// TIA Portal V16 export
// export: Created 2023-01-03T15:54:37.2222121Z, ExportSetting WithDefaults, DisplayName Totally Integrated Automation Portal, DisplayVersion V16, DisplayName TIA Portal Version Control Interface, DisplayVersion V16, DisplayName TIA Portal Openness, DisplayVersion V16, DisplayName STEP 7 Professional, DisplayVersion V16, DisplayName STEP 7 Safety, DisplayVersion V16, DisplayName WinCC Advanced, DisplayVersion V16
FUNCTION_BLOCK "MOTOR_AUTO"   // FB2, LAD
{ S7_Optimized_Access := 'TRUE' }
VERSION : 0.1
// stored: AutoNumber true, IsIECCheckEnabled false, IsRetainMemResEnabled false, MemoryReserve 100, SetENOAutomatically false, UDAEnableTagReadback false
   VAR_TEMP   // added for the SCL form of the ladder/FBD networks
      _w1 : Bool;
      _w2 : Bool;
   END_VAR
BEGIN

REGION Network 1: conveyor motor -M1 forwards fixed speed
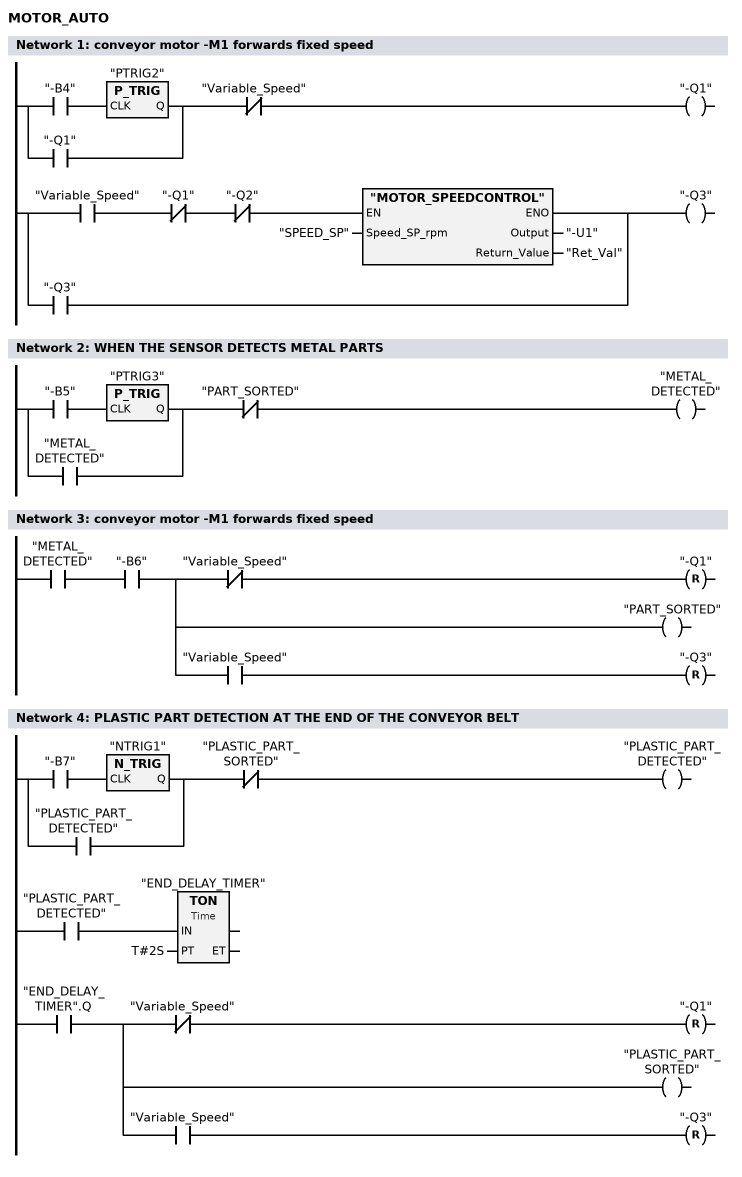
   RUNG wire#powerrail
      Contact( "-B4" )
      P_Trig( "PTRIG2" )
      wire#w1
      I_Contact( "Variable_Speed" )
      Coil( "-Q1" )
   END_RUNG
   RUNG wire#powerrail
      Contact( "-Q1" )
   END_RUNG wire#w1
   RUNG wire#powerrail
      Contact( "Variable_Speed" )
      I_Contact( "-Q1" )
      I_Contact( "-Q2" )
      "MOTOR_SPEEDCONTROL"(Speed_SP_rpm := "SPEED_SP", Output => "-U1", Return_Value => "Ret_Val")
      wire#w2
      Coil( "-Q3" )
   END_RUNG
   RUNG wire#powerrail
      Contact( "-Q3" )
   END_RUNG wire#w2
   // the same network as SCL:
   #_w1 := "-B4" AND NOT "PTRIG2";   // rising edge
   "PTRIG2" := "-B4";
   "-Q1" := (#_w1 OR "-Q1") AND NOT "Variable_Speed";
   "MOTOR_SPEEDCONTROL"(EN := "Variable_Speed" AND NOT "-Q1" AND NOT "-Q2",
                        Speed_SP_rpm := "SPEED_SP",
                        Output => "-U1",
                        Return_Value => "Ret_Val",
                        ENO => #_w2);
   "-Q3" := #_w2 OR "-Q3";
END_REGION

REGION Network 2: WHEN THE SENSOR DETECTS METAL PARTS
   RUNG wire#powerrail
      Contact( "-B5" )
      P_Trig( "PTRIG3" )
      wire#w1
      I_Contact( "PART_SORTED" )
      Coil( "METAL_DETECTED" )
   END_RUNG
   RUNG wire#powerrail
      Contact( "METAL_DETECTED" )
   END_RUNG wire#w1
   // the same network as SCL:
   #_w1 := "-B5" AND NOT "PTRIG3";   // rising edge
   "PTRIG3" := "-B5";
   "METAL_DETECTED" := (#_w1 OR "METAL_DETECTED") AND NOT "PART_SORTED";
END_REGION

REGION Network 3: conveyor motor -M1 forwards fixed speed
   RUNG wire#powerrail
      Contact( "METAL_DETECTED" )
      Contact( "-B6" )
      wire#w1
      I_Contact( "Variable_Speed" )
      R_Coil( "-Q1" )
   END_RUNG
   RUNG wire#w1
      Coil( "PART_SORTED" )
   END_RUNG
   RUNG wire#w1
      Contact( "Variable_Speed" )
      R_Coil( "-Q3" )
   END_RUNG
   // the same network as SCL:
   #_w1 := "METAL_DETECTED" AND "-B6";
   IF #_w1 AND NOT "Variable_Speed" THEN "-Q1" := FALSE; END_IF;
   "PART_SORTED" := #_w1;
   IF #_w1 AND "Variable_Speed" THEN "-Q3" := FALSE; END_IF;
END_REGION

REGION Network 4: PLASTIC PART DETECTION AT THE END OF THE CONVEYOR BELT
   RUNG wire#powerrail
      Contact( "-B7" )
      N_Trig( "NTRIG1" )
      wire#w1
      I_Contact( "PLASTIC_PART_SORTED" )
      Coil( "PLASTIC_PART_DETECTED" )
   END_RUNG
   RUNG wire#powerrail
      Contact( "PLASTIC_PART_DETECTED" )
   END_RUNG wire#w1
   RUNG wire#powerrail
      Contact( "PLASTIC_PART_DETECTED" )
      { S7_Templates := "time_type := Time" } "END_DELAY_TIMER".TON(pt := T#2S, et =>)
   END_RUNG
   RUNG wire#powerrail
      Contact( "END_DELAY_TIMER".Q )
      wire#w2
      I_Contact( "Variable_Speed" )
      R_Coil( "-Q1" )
   END_RUNG
   RUNG wire#w2
      Coil( "PLASTIC_PART_SORTED" )
   END_RUNG
   RUNG wire#w2
      Contact( "Variable_Speed" )
      R_Coil( "-Q3" )
   END_RUNG
   // the same network as SCL:
   #_w1 := NOT "-B7" AND "NTRIG1";   // falling edge
   "NTRIG1" := "-B7";
   "PLASTIC_PART_DETECTED" := (#_w1 OR "PLASTIC_PART_DETECTED") AND NOT "PLASTIC_PART_SORTED";
   "END_DELAY_TIMER".TON(IN := "PLASTIC_PART_DETECTED", PT := T#2S);
   IF "END_DELAY_TIMER".Q AND NOT "Variable_Speed" THEN "-Q1" := FALSE; END_IF;
   "PLASTIC_PART_SORTED" := "END_DELAY_TIMER".Q;
   IF "END_DELAY_TIMER".Q AND "Variable_Speed" THEN "-Q3" := FALSE; END_IF;
END_REGION
END_FUNCTION_BLOCK
